# B&R Automation Studio project HISTest (part 4)

```iecst
	SubBMS.Rack4.BSA.Rack_Calc.Field.BRA_Volt_Total 		:=	SHL(DWORD_TO_UINT(SHR(SubBMS.Rack4.BSA.Rack_Calc.Value[0], 8) AND 16#FF), 8) OR	DWORD_TO_UINT(SHR(SubBMS.Rack4.BSA.Rack_Calc.Value[0], 0) AND 16#FF);
	SubBMS.Rack4.BSA.Rack_Calc.Field.BRA_Curr_Total 		:=	SHL(DWORD_TO_UINT(SHR(SubBMS.Rack4.BSA.Rack_Calc.Value[0], 24) AND 16#FF), 8) OR	DWORD_TO_UINT(SHR(SubBMS.Rack4.BSA.Rack_Calc.Value[0], 16) AND 16#FF);
	SubBMS.Rack4.BSA.Rack_Calc.Field.BRA_SOC 				:=	SHL(DWORD_TO_UINT(SHR(SubBMS.Rack4.BSA.Rack_Calc.Value[1], 8) AND 16#FF), 8) OR	DWORD_TO_UINT(SHR(SubBMS.Rack4.BSA.Rack_Calc.Value[1], 0) AND 16#FF);
	SubBMS.Rack4.BSA.Rack_Calc.Field.BRA_SOH 				:=	SHL(DWORD_TO_UINT(SHR(SubBMS.Rack4.BSA.Rack_Calc.Value[1], 24) AND 16#FF), 8) OR	DWORD_TO_UINT(SHR(SubBMS.Rack4.BSA.Rack_Calc.Value[1], 16) AND 16#FF);

	SubBMS.Rack4.BSA.Rack_State.Field.BSA_Divice_Status 	:=	DWORD_TO_USINT(SHR(SubBMS.Rack4.BSA.Rack_State.Value[0], 0) AND 16#0F);
	SubBMS.Rack4.BSA.Rack_State.Field.BSA_Protect_Status 	:=	DWORD_TO_USINT(SHR(SubBMS.Rack4.BSA.Rack_State.Value[0], 8) AND 16#0F);
	SubBMS.Rack4.BSA.Rack_State.Field.BSA_Balance 			:=	SubBMS.Rack4.BSA.Rack_State.Value[0].16;
	SubBMS.Rack4.BSA.Rack_State.Field.BSA_Neg_Rly 			:=	SubBMS.Rack4.BSA.Rack_State.Value[0].17;
	SubBMS.Rack4.BSA.Rack_State.Field.BSA_Pos_Rly 			:=	SubBMS.Rack4.BSA.Rack_State.Value[0].18;
	SubBMS.Rack4.BSA.Rack_State.Field.BSA_PreChar_Rly 		:=	SubBMS.Rack4.BSA.Rack_State.Value[0].19;
	SubBMS.Rack4.BSA.Rack_State.Field.BSA_MSD_AUX 			:=	SubBMS.Rack4.BSA.Rack_State.Value[0].20;
	SubBMS.Rack4.BSA.Rack_State.Field.BSA_EMG_SW 			:=	SubBMS.Rack4.BSA.Rack_State.Value[0].21;
	SubBMS.Rack4.BSA.Rack_State.Field.BSA_Water_leak 		:=	SubBMS.Rack4.BSA.Rack_State.Value[0].22;
	SubBMS.Rack4.BSA.Rack_State.Field.Not_Used1 			:=	SubBMS.Rack4.BSA.Rack_State.Value[0].23;
	SubBMS.Rack4.BSA.Rack_State.Field.Not_Used2 			:=	DWORD_TO_USINT(SHR(SubBMS.Rack4.BSA.Rack_State.Value[0], 24) AND 16#0F);
	SubBMS.Rack4.BSA.Rack_State.Field.BSA_Ah 				:=	SHL(DWORD_TO_UINT(SHR(SubBMS.Rack4.BSA.Rack_State.Value[1], 8) AND 16#FF), 8) OR	DWORD_TO_UINT(SHR(SubBMS.Rack4.BSA.Rack_State.Value[1], 0) AND 16#FF);
	SubBMS.Rack4.BSA.Rack_State.Field.Not_Used3 			:=	SHL(DWORD_TO_UINT(SHR(SubBMS.Rack4.BSA.Rack_State.Value[1], 24) AND 16#FF), 8) OR DWORD_TO_UINT(SHR(SubBMS.Rack4.BSA.Rack_State.Value[1], 16) AND 16#FF);

	SubBMS.Rack4.BSA.Rack_AlarmState.Field.warning.BSA_Wn_Dischager_OC 			:= SubBMS.Rack4.BSA.Rack_AlarmState.Value[0].0;
	SubBMS.Rack4.BSA.Rack_AlarmState.Field.warning.BSA_Wn_Chager_OC				:= SubBMS.Rack4.BSA.Rack_AlarmState.Value[0].1;
	SubBMS.Rack4.BSA.Rack_AlarmState.Field.warning.BSA_Wn_SOC_OV 				:= SubBMS.Rack4.BSA.Rack_AlarmState.Value[0].2;
	SubBMS.Rack4.BSA.Rack_AlarmState.Field.warning.BSA_Wn_SOC_Un  				:= SubBMS.Rack4.BSA.Rack_AlarmState.Value[0].3;
	SubBMS.Rack4.BSA.Rack_AlarmState.Field.warning.BSA_Wn_OV  	 				:= SubBMS.Rack4.BSA.Rack_AlarmState.Value[0].4;
	SubBMS.Rack4.BSA.Rack_AlarmState.Field.warning.BSA_Wn_UV  		 			:= SubBMS.Rack4.BSA.Rack_AlarmState.Value[0].5;
	SubBMS.Rack4.BSA.Rack_AlarmState.Field.warning.BSA_Wn_Cell_OV  				:= SubBMS.Rack4.BSA.Rack_AlarmState.Value[0].6;
	SubBMS.Rack4.BSA.Rack_AlarmState.Field.warning.BSA_Wn_Cell_UV  				:= SubBMS.Rack4.BSA.Rack_AlarmState.Value[0].7;
	SubBMS.Rack4.BSA.Rack_AlarmState.Field.warning.BSA_Wn_Cell_UnbalV  			:= SubBMS.Rack4.BSA.Rack_AlarmState.Value[0].8;
	SubBMS.Rack4.BSA.Rack_AlarmState.Field.warning.BSA_Wn_DisCharger_Cell_OT 	:= SubBMS.Rack4.BSA.Rack_AlarmState.Value[0].9;
	SubBMS.Rack4.BSA.Rack_AlarmState.Field.warning.BSA_Wn_Charger_Cell_OT	 	:= SubBMS.Rack4.BSA.Rack_AlarmState.Value[0].10;
	SubBMS.Rack4.BSA.Rack_AlarmState.Field.warning.BSA_Wn_DisCharger_Cell_UT	:= SubBMS.Rack4.BSA.Rack_AlarmState.Value[0].11;
	SubBMS.Rack4.BSA.Rack_AlarmState.Field.warning.BSA_Wn_Charger_Cell_UT		:= SubBMS.Rack4.BSA.Rack_AlarmState.Value[0].12;
	SubBMS.Rack4.BSA.Rack_AlarmState.Field.warning.BSA_Wn_Cell_UnbalT 			:= SubBMS.Rack4.BSA.Rack_AlarmState.Value[0].13;
	SubBMS.Rack4.BSA.Rack_AlarmState.Field.warning.BSA_Wn_Discharger_UnbaPWR 	:= SubBMS.Rack4.BSA.Rack_AlarmState.Value[0].14;
	SubBMS.Rack4.BSA.Rack_AlarmState.Field.warning.BSA_Wn_Charger_UnbaPWR 		:= SubBMS.Rack4.BSA.Rack_AlarmState.Value[0].15;
	SubBMS.Rack4.BSA.Rack_AlarmState.Field.fault.BSA_FLT_Dischager_OC 			:= SubBMS.Rack4.BSA.Rack_AlarmState.Value[0].16;
	SubBMS.Rack4.BSA.Rack_AlarmState.Field.fault.BSA_FLT_Chager_OC 				:= SubBMS.Rack4.BSA.Rack_AlarmState.Value[0].17;
	SubBMS.Rack4.BSA.Rack_AlarmState.Field.fault.BSA_FLT_SOC_OV  				:= SubBMS.Rack4.BSA.Rack_AlarmState.Value[0].18;
	SubBMS.Rack4.BSA.Rack_AlarmState.Field.fault.BSA_FLT_SOC_Un  				:= SubBMS.Rack4.BSA.Rack_AlarmState.Value[0].19;
	SubBMS.Rack4.BSA.Rack_AlarmState.Field.fault.BSA_FLT_OV  					:= SubBMS.Rack4.BSA.Rack_AlarmState.Value[0].20;
	SubBMS.Rack4.BSA.Rack_AlarmState.Field.fault.BSA_FLT_UV  					:= SubBMS.Rack4.BSA.Rack_AlarmState.Value[0].21;
	SubBMS.Rack4.BSA.Rack_AlarmState.Field.fault.BSA_FLT_Cell_OV  				:= SubBMS.Rack4.BSA.Rack_AlarmState.Value[0].22;
	SubBMS.Rack4.BSA.Rack_AlarmState.Field.fault.BSA_FLT_Cell_UV  				:= SubBMS.Rack4.BSA.Rack_AlarmState.Value[0].23;
	SubBMS.Rack4.BSA.Rack_AlarmState.Field.fault.BSA_FLT_Cell_UnbalV 			:= SubBMS.Rack4.BSA.Rack_AlarmState.Value[0].24;
	SubBMS.Rack4.BSA.Rack_AlarmState.Field.fault.BSA_FLT_DisCharger_Cell_OT  	:= SubBMS.Rack4.BSA.Rack_AlarmState.Value[0].25;
	SubBMS.Rack4.BSA.Rack_AlarmState.Field.fault.BSA_FLT_Charger_Cell_OT  		:= SubBMS.Rack4.BSA.Rack_AlarmState.Value[0].26;
	SubBMS.Rack4.BSA.Rack_AlarmState.Field.fault.BSA_FLT_DisCharger_Cell_UT 	:= SubBMS.Rack4.BSA.Rack_AlarmState.Value[0].27;
	SubBMS.Rack4.BSA.Rack_AlarmState.Field.fault.BSA_FLT_Charger_Cell_UT  		:= SubBMS.Rack4.BSA.Rack_AlarmState.Value[0].28;
	SubBMS.Rack4.BSA.Rack_AlarmState.Field.fault.BSA_FLT_Cell_UnbalT  			:= SubBMS.Rack4.BSA.Rack_AlarmState.Value[0].29;
	SubBMS.Rack4.BSA.Rack_AlarmState.Field.fault.BSA_FLT_Discharger_UnbaPWR  	:= SubBMS.Rack4.BSA.Rack_AlarmState.Value[0].30;
	SubBMS.Rack4.BSA.Rack_AlarmState.Field.fault.BSA_FLT_Charger_UnbaPWR  		:= SubBMS.Rack4.BSA.Rack_AlarmState.Value[0].31;
	SubBMS.Rack4.BSA.Rack_AlarmState.Field.protect.BSA_Prtct_Dischager_OC   	:= SubBMS.Rack4.BSA.Rack_AlarmState.Value[1].0;
	SubBMS.Rack4.BSA.Rack_AlarmState.Field.protect.BSA_Prtct_Chager_OC   		:= SubBMS.Rack4.BSA.Rack_AlarmState.Value[1].1;
	SubBMS.Rack4.BSA.Rack_AlarmState.Field.protect.BSA_Prtct_SOC_OV   		  	:= SubBMS.Rack4.BSA.Rack_AlarmState.Value[1].2;
	SubBMS.Rack4.BSA.Rack_AlarmState.Field.protect.BSA_Prtct_SOC_Un   		  	:= SubBMS.Rack4.BSA.Rack_AlarmState.Value[1].3;
	SubBMS.Rack4.BSA.Rack_AlarmState.Field.protect.BSA_Prtct_OV   		  		:= SubBMS.Rack4.BSA.Rack_AlarmState.Value[1].4;
	SubBMS.Rack4.BSA.Rack_AlarmState.Field.protect.BSA_Prtct_UV   		  		:= SubBMS.Rack4.BSA.Rack_AlarmState.Value[1].5;
	SubBMS.Rack4.BSA.Rack_AlarmState.Field.protect.BSA_Prtct_Cell_OV   		  	:= SubBMS.Rack4.BSA.Rack_AlarmState.Value[1].6;
	SubBMS.Rack4.BSA.Rack_AlarmState.Field.protect.BSA_Prtct_Cell_UV   		  	:= SubBMS.Rack4.BSA.Rack_AlarmState.Value[1].7;
	SubBMS.Rack4.BSA.Rack_AlarmState.Field.protect.BSA_Prtct_Cell_UnbalV   		:= SubBMS.Rack4.BSA.Rack_AlarmState.Value[1].8;
	SubBMS.Rack4.BSA.Rack_AlarmState.Field.protect.BSA_Prtct_DisCharger_Cell_OT := SubBMS.Rack4.BSA.Rack_AlarmState.Value[1].9;
	SubBMS.Rack4.BSA.Rack_AlarmState.Field.protect.BSA_Prtct_Charger_Cell_OT 	:= SubBMS.Rack4.BSA.Rack_AlarmState.Value[1].10;
	SubBMS.Rack4.BSA.Rack_AlarmState.Field.protect.BSA_Prtct_DisCharger_Cell_UT := SubBMS.Rack4.BSA.Rack_AlarmState.Value[1].11;
	SubBMS.Rack4.BSA.Rack_AlarmState.Field.protect.BSA_Prtct_Charger_Cell_UT   	:= SubBMS.Rack4.BSA.Rack_AlarmState.Value[1].12;
	SubBMS.Rack4.BSA.Rack_AlarmState.Field.protect.BSA_Prtct_Cell_UnbalT   		:= SubBMS.Rack4.BSA.Rack_AlarmState.Value[1].13;
	SubBMS.Rack4.BSA.Rack_AlarmState.Field.protect.BSA_Prtct_Discharger_UnbaPWR := SubBMS.Rack4.BSA.Rack_AlarmState.Value[1].14;
	SubBMS.Rack4.BSA.Rack_AlarmState.Field.protect.BSA_Prtct_Charger_UnbaPWR   	:= SubBMS.Rack4.BSA.Rack_AlarmState.Value[1].15;
	SubBMS.Rack4.BSA.Rack_AlarmState.Field.protect.BSA_Prtct_Rly_Err   			:= SubBMS.Rack4.BSA.Rack_AlarmState.Value[1].16;
	SubBMS.Rack4.BSA.Rack_AlarmState.Field.protect.BSA_Prtct_IN_COM_Err   		:= SubBMS.Rack4.BSA.Rack_AlarmState.Value[1].17;
	SubBMS.Rack4.BSA.Rack_AlarmState.Field.protect.BSA_Prtct_EX_COM_Err   		:= SubBMS.Rack4.BSA.Rack_AlarmState.Value[1].18;
	SubBMS.Rack4.BSA.Rack_AlarmState.Field.protect.BSA_Prtct_CT_COM_Err   		:= SubBMS.Rack4.BSA.Rack_AlarmState.Value[1].19;
	SubBMS.Rack4.BSA.Rack_AlarmState.Field.protect.BSA_Prtct_Water_Leak_Err   	:= SubBMS.Rack4.BSA.Rack_AlarmState.Value[1].20;
	SubBMS.Rack4.BSA.Rack_AlarmState.Field.protect.BSA_Prtct_EMS_SW_Err  		:= SubBMS.Rack4.BSA.Rack_AlarmState.Value[1].21;
	SubBMS.Rack4.BSA.Rack_AlarmState.Field.protect.Not_Used1 					:= SubBMS.Rack4.BSA.Rack_AlarmState.Value[1].22;
	SubBMS.Rack4.BSA.Rack_AlarmState.Field.protect.Not_Used2 					:= SubBMS.Rack4.BSA.Rack_AlarmState.Value[1].23;
	SubBMS.Rack4.BSA.Rack_AlarmState.Field.protect.Not_Used3 					:= DWORD_TO_USINT(SHR(SubBMS.Rack4.BSA.Rack_AlarmState.Value[1], 24) AND 16#0F);

	SubBMS.Rack4.BSA.Rack_PWRCalc.Field.BSA_CHAPWCont 							:=	SHL(DWORD_TO_UINT(SHR(SubBMS.Rack4.BSA.Rack_PWRCalc.Value[0], 8) AND 16#FF), 8) OR	DWORD_TO_UINT(SHR(SubBMS.Rack4.BSA.Rack_PWRCalc.Value[0], 0) AND 16#FF);
	SubBMS.Rack4.BSA.Rack_PWRCalc.Field.BSA_DisCHAPWCont 						:=	SHL(DWORD_TO_UINT(SHR(SubBMS.Rack4.BSA.Rack_PWRCalc.Value[0], 24) AND 16#FF), 8) OR	DWORD_TO_UINT(SHR(SubBMS.Rack4.BSA.Rack_PWRCalc.Value[0], 16) AND 16#FF);
	SubBMS.Rack4.BSA.Rack_PWRCalc.Field.BSA_CHAPWPeak 							:=	SHL(DWORD_TO_UINT(SHR(SubBMS.Rack4.BSA.Rack_PWRCalc.Value[1], 8) AND 16#FF), 8) OR	DWORD_TO_UINT(SHR(SubBMS.Rack4.BSA.Rack_PWRCalc.Value[1], 0) AND 16#FF);
	SubBMS.Rack4.BSA.Rack_PWRCalc.Field.BSA_DisCHAPWPeak 						:=	SHL(DWORD_TO_UINT(SHR(SubBMS.Rack4.BSA.Rack_PWRCalc.Value[1], 24) AND 16#FF), 8) OR	DWORD_TO_UINT(SHR(SubBMS.Rack4.BSA.Rack_PWRCalc.Value[1], 16) AND 16#FF);

	SubBMS.Rack4.BSA.Rack_Cell_Vcalc.Field.BSA_Cell_MaxV 						:=	SHL(DWORD_TO_UINT(SHR(SubBMS.Rack4.BSA.Rack_Cell_Vcalc.Value[0], 8) AND 16#FF), 8) OR	DWORD_TO_UINT(SHR(SubBMS.Rack4.BSA.Rack_Cell_Vcalc.Value[0], 0) AND 16#FF);
	SubBMS.Rack4.BSA.Rack_Cell_Vcalc.Field.BSA_Cell_MinV 						:=	SHL(DWORD_TO_UINT(SHR(SubBMS.Rack4.BSA.Rack_Cell_Vcalc.Value[0], 24) AND 16#FF), 8) OR	DWORD_TO_UINT(SHR(SubBMS.Rack4.BSA.Rack_Cell_Vcalc.Value[0], 16) AND 16#FF);
	SubBMS.Rack4.BSA.Rack_Cell_Vcalc.Field.BSA_Cell_AVGV 						:=	SHL(DWORD_TO_UINT(SHR(SubBMS.Rack4.BSA.Rack_Cell_Vcalc.Value[1], 8) AND 16#FF), 8) OR	DWORD_TO_UINT(SHR(SubBMS.Rack4.BSA.Rack_Cell_Vcalc.Value[1], 0) AND 16#FF);
	SubBMS.Rack4.BSA.Rack_Cell_Vcalc.Field.BSA_Cell_DeviV 						:=	SHL(DWORD_TO_UINT(SHR(SubBMS.Rack4.BSA.Rack_Cell_Vcalc.Value[1], 24) AND 16#FF), 8) OR	DWORD_TO_UINT(SHR(SubBMS.Rack4.BSA.Rack_Cell_Vcalc.Value[1], 16) AND 16#FF);

	SubBMS.Rack4.BSA.Rack_Cell_Tcalc.Field.BSA_Cell_MaxT 						:=	SHL(DWORD_TO_UINT(SHR(SubBMS.Rack4.BSA.Rack_Cell_Tcalc.Value[0], 8) AND 16#FF), 8) OR	DWORD_TO_UINT(SHR(SubBMS.Rack4.BSA.Rack_Cell_Tcalc.Value[0], 0) AND 16#FF);
	SubBMS.Rack4.BSA.Rack_Cell_Tcalc.Field.BSA_Cell_MinT 						:=	SHL(DWORD_TO_UINT(SHR(SubBMS.Rack4.BSA.Rack_Cell_Tcalc.Value[0], 24) AND 16#FF), 8) OR	DWORD_TO_UINT(SHR(SubBMS.Rack4.BSA.Rack_Cell_Tcalc.Value[0], 16) AND 16#FF);
	SubBMS.Rack4.BSA.Rack_Cell_Tcalc.Field.BSA_Cell_AVGT 						:=	SHL(DWORD_TO_UINT(SHR(SubBMS.Rack4.BSA.Rack_Cell_Tcalc.Value[1], 8) AND 16#FF), 8) OR	DWORD_TO_UINT(SHR(SubBMS.Rack4.BSA.Rack_Cell_Tcalc.Value[1], 0) AND 16#FF);
	SubBMS.Rack4.BSA.Rack_Cell_Tcalc.Field.BSA_Cell_DeviT 						:=	SHL(DWORD_TO_UINT(SHR(SubBMS.Rack4.BSA.Rack_Cell_Tcalc.Value[1], 24) AND 16#FF), 8) OR	DWORD_TO_UINT(SHR(SubBMS.Rack4.BSA.Rack_Cell_Tcalc.Value[1], 16) AND 16#FF);

	SubBMS.Rack4.BSA.Rack_Cell_Pcalc.Field.BSA_Cell_MaxV_Location 				:=	SHL(DWORD_TO_UINT(SHR(SubBMS.Rack4.BSA.Rack_Cell_Pcalc.Value[0], 8) AND 16#FF), 8) OR	DWORD_TO_UINT(SHR(SubBMS.Rack4.BSA.Rack_Cell_Pcalc.Value[0], 0) AND 16#FF);
	SubBMS.Rack4.BSA.Rack_Cell_Pcalc.Field.BSA_Cell_MinV_Location 				:=	SHL(DWORD_TO_UINT(SHR(SubBMS.Rack4.BSA.Rack_Cell_Pcalc.Value[0], 24) AND 16#FF), 8) OR	DWORD_TO_UINT(SHR(SubBMS.Rack4.BSA.Rack_Cell_Pcalc.Value[0], 16) AND 16#FF);
	SubBMS.Rack4.BSA.Rack_Cell_Pcalc.Field.BSA_Cell_MaxT_Location 				:=	SHL(DWORD_TO_UINT(SHR(SubBMS.Rack4.BSA.Rack_Cell_Pcalc.Value[1], 8) AND 16#FF), 8) OR	DWORD_TO_UINT(SHR(SubBMS.Rack4.BSA.Rack_Cell_Pcalc.Value[1], 0) AND 16#FF);
	SubBMS.Rack4.BSA.Rack_Cell_Pcalc.Field.BSA_Cell_MinT_Location 				:=	SHL(DWORD_TO_UINT(SHR(SubBMS.Rack4.BSA.Rack_Cell_Pcalc.Value[1], 24) AND 16#FF), 8) OR	DWORD_TO_UINT(SHR(SubBMS.Rack4.BSA.Rack_Cell_Pcalc.Value[1], 16) AND 16#FF);

	SubBMS.Rack4.BSA.Modul1_Info.Field.Volt_Total 								:=	SHL(DWORD_TO_UINT(SHR(SubBMS.Rack4.BSA.Modul1_Info.Value[0], 8) AND 16#FF), 8) OR	DWORD_TO_UINT(SHR(SubBMS.Rack4.BSA.Modul1_Info.Value[0], 0) AND 16#FF);
	SubBMS.Rack4.BSA.Modul1_Info.Field.Agv_Volt 								:=	SHL(DWORD_TO_UINT(SHR(SubBMS.Rack4.BSA.Modul1_Info.Value[0], 24) AND 16#FF), 8) OR	DWORD_TO_UINT(SHR(SubBMS.Rack4.BSA.Modul1_Info.Value[0], 16) AND 16#FF);
	SubBMS.Rack4.BSA.Modul1_Info.Field.Agv_Temp 								:=	SHL(DWORD_TO_UINT(SHR(SubBMS.Rack4.BSA.Modul1_Info.Value[1], 8) AND 16#FF), 8) OR	DWORD_TO_UINT(SHR(SubBMS.Rack4.BSA.Modul1_Info.Value[1], 0) AND 16#FF);
	SubBMS.Rack4.BSA.Modul1_Info.Field.OPS_INITOK 								:= SubBMS.Rack4.BSA.Modul1_Info.Value[1].16;
	SubBMS.Rack4.BSA.Modul1_Info.Field.OPS_Fault  								:= SubBMS.Rack4.BSA.Modul1_Info.Value[1].17;
	SubBMS.Rack4.BSA.Modul1_Info.Field.OPS_Balan_On_OFF  						:= SubBMS.Rack4.BSA.Modul1_Info.Value[1].18;
	SubBMS.Rack4.BSA.Modul1_Info.Field.OPS_Waterleak_Err  						:= SubBMS.Rack4.BSA.Modul1_Info.Value[1].19;
	SubBMS.Rack4.BSA.Modul1_Info.Field.OPS_CellVolt_Err  						:= SubBMS.Rack4.BSA.Modul1_Info.Value[1].20;
	SubBMS.Rack4.BSA.Modul1_Info.Field.OPS_CellTemps_Err  						:= SubBMS.Rack4.BSA.Modul1_Info.Value[1].21;
	SubBMS.Rack4.BSA.Modul1_Info.Field.BATIC_Err  								:= SubBMS.Rack4.BSA.Modul1_Info.Value[1].22;
	SubBMS.Rack4.BSA.Modul1_Info.Field.CTCOM_Err  								:= SubBMS.Rack4.BSA.Modul1_Info.Value[1].23;
	SubBMS.Rack4.BSA.Modul1_Info.Field.OPS_MBCOM_Err  							:= SubBMS.Rack4.BSA.Modul1_Info.Value[1].24;
	SubBMS.Rack4.BSA.Modul1_Info.Field.Not_Used1 								:= SubBMS.Rack4.BSA.Modul1_Info.Value[1].25;
	SubBMS.Rack4.BSA.Modul1_Info.Field.Not_Used2  								:= SubBMS.Rack4.BSA.Modul1_Info.Value[1].26;
	SubBMS.Rack4.BSA.Modul1_Info.Field.Not_Used3  								:= SubBMS.Rack4.BSA.Modul1_Info.Value[1].27;
	SubBMS.Rack4.BSA.Modul1_Info.Field.Not_Used4  								:= SubBMS.Rack4.BSA.Modul1_Info.Value[1].28;
	SubBMS.Rack4.BSA.Modul1_Info.Field.Not_Used5  								:= SubBMS.Rack4.BSA.Modul1_Info.Value[1].29;
	SubBMS.Rack4.BSA.Modul1_Info.Field.Not_Used6  								:= SubBMS.Rack4.BSA.Modul1_Info.Value[1].30;
	SubBMS.Rack4.BSA.Modul1_Info.Field.Not_Used7  								:= SubBMS.Rack4.BSA.Modul1_Info.Value[1].31;

	SubBMS.Rack4.BSA.Modul2_Info.Field.Volt_Total 								:=	SHL(DWORD_TO_UINT(SHR(SubBMS.Rack4.BSA.Modul2_Info.Value[0], 8) AND 16#FF), 8) OR	DWORD_TO_UINT(SHR(SubBMS.Rack4.BSA.Modul2_Info.Value[0], 0) AND 16#FF);
	SubBMS.Rack4.BSA.Modul2_Info.Field.Agv_Volt 								:=	SHL(DWORD_TO_UINT(SHR(SubBMS.Rack4.BSA.Modul2_Info.Value[0], 24) AND 16#FF), 8) OR	DWORD_TO_UINT(SHR(SubBMS.Rack4.BSA.Modul2_Info.Value[0], 16) AND 16#FF);
	SubBMS.Rack4.BSA.Modul2_Info.Field.Agv_Temp 								:=	SHL(DWORD_TO_UINT(SHR(SubBMS.Rack4.BSA.Modul2_Info.Value[1], 8) AND 16#FF), 8) OR	DWORD_TO_UINT(SHR(SubBMS.Rack4.BSA.Modul2_Info.Value[1], 0) AND 16#FF);
	SubBMS.Rack4.BSA.Modul2_Info.Field.OPS_INITOK 								:= SubBMS.Rack4.BSA.Modul2_Info.Value[1].16;
	SubBMS.Rack4.BSA.Modul2_Info.Field.OPS_Fault  								:= SubBMS.Rack4.BSA.Modul2_Info.Value[1].17;
	SubBMS.Rack4.BSA.Modul2_Info.Field.OPS_Balan_On_OFF  						:= SubBMS.Rack4.BSA.Modul2_Info.Value[1].18;
	SubBMS.Rack4.BSA.Modul2_Info.Field.OPS_Waterleak_Err  						:= SubBMS.Rack4.BSA.Modul2_Info.Value[1].19;
	SubBMS.Rack4.BSA.Modul2_Info.Field.OPS_CellVolt_Err  						:= SubBMS.Rack4.BSA.Modul2_Info.Value[1].20;
	SubBMS.Rack4.BSA.Modul2_Info.Field.OPS_CellTemps_Err  						:= SubBMS.Rack4.BSA.Modul2_Info.Value[1].21;
	SubBMS.Rack4.BSA.Modul2_Info.Field.BATIC_Err  								:= SubBMS.Rack4.BSA.Modul2_Info.Value[1].22;
	SubBMS.Rack4.BSA.Modul2_Info.Field.CTCOM_Err  								:= SubBMS.Rack4.BSA.Modul2_Info.Value[1].23;
	SubBMS.Rack4.BSA.Modul2_Info.Field.OPS_MBCOM_Err  							:= SubBMS.Rack4.BSA.Modul2_Info.Value[1].24;
	SubBMS.Rack4.BSA.Modul2_Info.Field.Not_Used1 								:= SubBMS.Rack4.BSA.Modul2_Info.Value[1].25;
	SubBMS.Rack4.BSA.Modul2_Info.Field.Not_Used2  								:= SubBMS.Rack4.BSA.Modul2_Info.Value[1].26;
	SubBMS.Rack4.BSA.Modul2_Info.Field.Not_Used3  								:= SubBMS.Rack4.BSA.Modul2_Info.Value[1].27;
	SubBMS.Rack4.BSA.Modul2_Info.Field.Not_Used4  								:= SubBMS.Rack4.BSA.Modul2_Info.Value[1].28;
	SubBMS.Rack4.BSA.Modul2_Info.Field.Not_Used5  								:= SubBMS.Rack4.BSA.Modul2_Info.Value[1].29;
	SubBMS.Rack4.BSA.Modul2_Info.Field.Not_Used6  								:= SubBMS.Rack4.BSA.Modul2_Info.Value[1].30;
	SubBMS.Rack4.BSA.Modul2_Info.Field.Not_Used7  								:= SubBMS.Rack4.BSA.Modul2_Info.Value[1].31;

	SubBMS.Rack4.BSA.Modul3_Info.Field.Volt_Total 								:=	SHL(DWORD_TO_UINT(SHR(SubBMS.Rack4.BSA.Modul3_Info.Value[0], 8) AND 16#FF), 8) OR	DWORD_TO_UINT(SHR(SubBMS.Rack4.BSA.Modul3_Info.Value[0], 0) AND 16#FF);
	SubBMS.Rack4.BSA.Modul3_Info.Field.Agv_Volt 								:=	SHL(DWORD_TO_UINT(SHR(SubBMS.Rack4.BSA.Modul3_Info.Value[0], 24) AND 16#FF), 8) OR	DWORD_TO_UINT(SHR(SubBMS.Rack4.BSA.Modul3_Info.Value[0], 16) AND 16#FF);
	SubBMS.Rack4.BSA.Modul3_Info.Field.Agv_Temp 								:=	SHL(DWORD_TO_UINT(SHR(SubBMS.Rack4.BSA.Modul3_Info.Value[1], 8) AND 16#FF), 8) OR	DWORD_TO_UINT(SHR(SubBMS.Rack4.BSA.Modul3_Info.Value[1], 0) AND 16#FF);
	SubBMS.Rack4.BSA.Modul3_Info.Field.OPS_INITOK 								:= SubBMS.Rack4.BSA.Modul3_Info.Value[1].16;
	SubBMS.Rack4.BSA.Modul3_Info.Field.OPS_Fault  								:= SubBMS.Rack4.BSA.Modul3_Info.Value[1].17;
	SubBMS.Rack4.BSA.Modul3_Info.Field.OPS_Balan_On_OFF  						:= SubBMS.Rack4.BSA.Modul3_Info.Value[1].18;
	SubBMS.Rack4.BSA.Modul3_Info.Field.OPS_Waterleak_Err  						:= SubBMS.Rack4.BSA.Modul3_Info.Value[1].19;
	SubBMS.Rack4.BSA.Modul3_Info.Field.OPS_CellVolt_Err  						:= SubBMS.Rack4.BSA.Modul3_Info.Value[1].20;
	SubBMS.Rack4.BSA.Modul3_Info.Field.OPS_CellTemps_Err  						:= SubBMS.Rack4.BSA.Modul3_Info.Value[1].21;
	SubBMS.Rack4.BSA.Modul3_Info.Field.BATIC_Err  								:= SubBMS.Rack4.BSA.Modul3_Info.Value[1].22;
	SubBMS.Rack4.BSA.Modul3_Info.Field.CTCOM_Err  								:= SubBMS.Rack4.BSA.Modul3_Info.Value[1].23;
	SubBMS.Rack4.BSA.Modul3_Info.Field.OPS_MBCOM_Err  							:= SubBMS.Rack4.BSA.Modul3_Info.Value[1].24;
	SubBMS.Rack4.BSA.Modul3_Info.Field.Not_Used1 								:= SubBMS.Rack4.BSA.Modul3_Info.Value[1].25;
	SubBMS.Rack4.BSA.Modul3_Info.Field.Not_Used2  								:= SubBMS.Rack4.BSA.Modul3_Info.Value[1].26;
	SubBMS.Rack4.BSA.Modul3_Info.Field.Not_Used3  								:= SubBMS.Rack4.BSA.Modul3_Info.Value[1].27;
	SubBMS.Rack4.BSA.Modul3_Info.Field.Not_Used4  								:= SubBMS.Rack4.BSA.Modul3_Info.Value[1].28;
	SubBMS.Rack4.BSA.Modul3_Info.Field.Not_Used5  								:= SubBMS.Rack4.BSA.Modul3_Info.Value[1].29;
	SubBMS.Rack4.BSA.Modul3_Info.Field.Not_Used6  								:= SubBMS.Rack4.BSA.Modul3_Info.Value[1].30;
	SubBMS.Rack4.BSA.Modul3_Info.Field.Not_Used7  								:= SubBMS.Rack4.BSA.Modul3_Info.Value[1].31;

	SubBMS.Rack4.BSA.Modul4_Info.Field.Volt_Total 								:=	SHL(DWORD_TO_UINT(SHR(SubBMS.Rack4.BSA.Modul4_Info.Value[0], 8) AND 16#FF), 8) OR	DWORD_TO_UINT(SHR(SubBMS.Rack4.BSA.Modul4_Info.Value[0], 0) AND 16#FF);
	SubBMS.Rack4.BSA.Modul4_Info.Field.Agv_Volt 								:=	SHL(DWORD_TO_UINT(SHR(SubBMS.Rack4.BSA.Modul4_Info.Value[0], 24) AND 16#FF), 8) OR	DWORD_TO_UINT(SHR(SubBMS.Rack4.BSA.Modul4_Info.Value[0], 16) AND 16#FF);
	SubBMS.Rack4.BSA.Modul4_Info.Field.Agv_Temp 								:=	SHL(DWORD_TO_UINT(SHR(SubBMS.Rack4.BSA.Modul4_Info.Value[1], 8) AND 16#FF), 8) OR	DWORD_TO_UINT(SHR(SubBMS.Rack4.BSA.Modul4_Info.Value[1], 0) AND 16#FF);
	SubBMS.Rack4.BSA.Modul4_Info.Field.OPS_INITOK 								:= SubBMS.Rack4.BSA.Modul4_Info.Value[1].16;
	SubBMS.Rack4.BSA.Modul4_Info.Field.OPS_Fault  								:= SubBMS.Rack4.BSA.Modul4_Info.Value[1].17;
	SubBMS.Rack4.BSA.Modul4_Info.Field.OPS_Balan_On_OFF  						:= SubBMS.Rack4.BSA.Modul4_Info.Value[1].18;
	SubBMS.Rack4.BSA.Modul4_Info.Field.OPS_Waterleak_Err  						:= SubBMS.Rack4.BSA.Modul4_Info.Value[1].19;
	SubBMS.Rack4.BSA.Modul4_Info.Field.OPS_CellVolt_Err  						:= SubBMS.Rack4.BSA.Modul4_Info.Value[1].20;
	SubBMS.Rack4.BSA.Modul4_Info.Field.OPS_CellTemps_Err  						:= SubBMS.Rack4.BSA.Modul4_Info.Value[1].21;
	SubBMS.Rack4.BSA.Modul4_Info.Field.BATIC_Err  								:= SubBMS.Rack4.BSA.Modul4_Info.Value[1].22;
	SubBMS.Rack4.BSA.Modul4_Info.Field.CTCOM_Err  								:= SubBMS.Rack4.BSA.Modul4_Info.Value[1].23;
	SubBMS.Rack4.BSA.Modul4_Info.Field.OPS_MBCOM_Err  							:= SubBMS.Rack4.BSA.Modul4_Info.Value[1].24;
	SubBMS.Rack4.BSA.Modul4_Info.Field.Not_Used1 								:= SubBMS.Rack4.BSA.Modul4_Info.Value[1].25;
	SubBMS.Rack4.BSA.Modul4_Info.Field.Not_Used2  								:= SubBMS.Rack4.BSA.Modul4_Info.Value[1].26;
	SubBMS.Rack4.BSA.Modul4_Info.Field.Not_Used3  								:= SubBMS.Rack4.BSA.Modul4_Info.Value[1].27;
	SubBMS.Rack4.BSA.Modul4_Info.Field.Not_Used4  								:= SubBMS.Rack4.BSA.Modul4_Info.Value[1].28;
	SubBMS.Rack4.BSA.Modul4_Info.Field.Not_Used5  								:= SubBMS.Rack4.BSA.Modul4_Info.Value[1].29;
	SubBMS.Rack4.BSA.Modul4_Info.Field.Not_Used6  								:= SubBMS.Rack4.BSA.Modul4_Info.Value[1].30;
	SubBMS.Rack4.BSA.Modul4_Info.Field.Not_Used7  								:= SubBMS.Rack4.BSA.Modul4_Info.Value[1].31;

	SubBMS.Rack4.BSA.Modul5_Info.Field.Volt_Total 								:=	SHL(DWORD_TO_UINT(SHR(SubBMS.Rack4.BSA.Modul5_Info.Value[0], 8) AND 16#FF), 8) OR	DWORD_TO_UINT(SHR(SubBMS.Rack4.BSA.Modul5_Info.Value[0], 0) AND 16#FF);
	SubBMS.Rack4.BSA.Modul5_Info.Field.Agv_Volt 								:=	SHL(DWORD_TO_UINT(SHR(SubBMS.Rack4.BSA.Modul5_Info.Value[0], 24) AND 16#FF), 8) OR	DWORD_TO_UINT(SHR(SubBMS.Rack4.BSA.Modul5_Info.Value[0], 16) AND 16#FF);
	SubBMS.Rack4.BSA.Modul5_Info.Field.Agv_Temp 								:=	SHL(DWORD_TO_UINT(SHR(SubBMS.Rack4.BSA.Modul5_Info.Value[1], 8) AND 16#FF), 8) OR	DWORD_TO_UINT(SHR(SubBMS.Rack4.BSA.Modul5_Info.Value[1], 0) AND 16#FF);
	SubBMS.Rack4.BSA.Modul5_Info.Field.OPS_INITOK 								:= SubBMS.Rack4.BSA.Modul5_Info.Value[1].16;
	SubBMS.Rack4.BSA.Modul5_Info.Field.OPS_Fault  								:= SubBMS.Rack4.BSA.Modul5_Info.Value[1].17;
	SubBMS.Rack4.BSA.Modul5_Info.Field.OPS_Balan_On_OFF  						:= SubBMS.Rack4.BSA.Modul5_Info.Value[1].18;
	SubBMS.Rack4.BSA.Modul5_Info.Field.OPS_Waterleak_Err  						:= SubBMS.Rack4.BSA.Modul5_Info.Value[1].19;
	SubBMS.Rack4.BSA.Modul5_Info.Field.OPS_CellVolt_Err  						:= SubBMS.Rack4.BSA.Modul5_Info.Value[1].20;
	SubBMS.Rack4.BSA.Modul5_Info.Field.OPS_CellTemps_Err  						:= SubBMS.Rack4.BSA.Modul5_Info.Value[1].21;
	SubBMS.Rack4.BSA.Modul5_Info.Field.BATIC_Err  								:= SubBMS.Rack4.BSA.Modul5_Info.Value[1].22;
	SubBMS.Rack4.BSA.Modul5_Info.Field.CTCOM_Err  								:= SubBMS.Rack4.BSA.Modul5_Info.Value[1].23;
	SubBMS.Rack4.BSA.Modul5_Info.Field.OPS_MBCOM_Err  							:= SubBMS.Rack4.BSA.Modul5_Info.Value[1].24;
	SubBMS.Rack4.BSA.Modul5_Info.Field.Not_Used1 								:= SubBMS.Rack4.BSA.Modul5_Info.Value[1].25;
	SubBMS.Rack4.BSA.Modul5_Info.Field.Not_Used2  								:= SubBMS.Rack4.BSA.Modul5_Info.Value[1].26;
	SubBMS.Rack4.BSA.Modul5_Info.Field.Not_Used3  								:= SubBMS.Rack4.BSA.Modul5_Info.Value[1].27;
	SubBMS.Rack4.BSA.Modul5_Info.Field.Not_Used4  								:= SubBMS.Rack4.BSA.Modul5_Info.Value[1].28;
	SubBMS.Rack4.BSA.Modul5_Info.Field.Not_Used5  								:= SubBMS.Rack4.BSA.Modul5_Info.Value[1].29;
	SubBMS.Rack4.BSA.Modul5_Info.Field.Not_Used6  								:= SubBMS.Rack4.BSA.Modul5_Info.Value[1].30;
	SubBMS.Rack4.BSA.Modul5_Info.Field.Not_Used7  								:= SubBMS.Rack4.BSA.Modul5_Info.Value[1].31;

	SubBMS.Rack4.BSA.Modul6_Info.Field.Volt_Total 								:=	SHL(DWORD_TO_UINT(SHR(SubBMS.Rack4.BSA.Modul6_Info.Value[0], 8) AND 16#FF), 8) OR	DWORD_TO_UINT(SHR(SubBMS.Rack4.BSA.Modul6_Info.Value[0], 0) AND 16#FF);
	SubBMS.Rack4.BSA.Modul6_Info.Field.Agv_Volt 								:=	SHL(DWORD_TO_UINT(SHR(SubBMS.Rack4.BSA.Modul6_Info.Value[0], 24) AND 16#FF), 8) OR	DWORD_TO_UINT(SHR(SubBMS.Rack4.BSA.Modul6_Info.Value[0], 16) AND 16#FF);
	SubBMS.Rack4.BSA.Modul6_Info.Field.Agv_Temp 								:=	SHL(DWORD_TO_UINT(SHR(SubBMS.Rack4.BSA.Modul6_Info.Value[1], 8) AND 16#FF), 8) OR	DWORD_TO_UINT(SHR(SubBMS.Rack4.BSA.Modul6_Info.Value[1], 0) AND 16#FF);
	SubBMS.Rack4.BSA.Modul6_Info.Field.OPS_INITOK 								:= SubBMS.Rack4.BSA.Modul6_Info.Value[1].16;
	SubBMS.Rack4.BSA.Modul6_Info.Field.OPS_Fault  								:= SubBMS.Rack4.BSA.Modul6_Info.Value[1].17;
	SubBMS.Rack4.BSA.Modul6_Info.Field.OPS_Balan_On_OFF  						:= SubBMS.Rack4.BSA.Modul6_Info.Value[1].18;
	SubBMS.Rack4.BSA.Modul6_Info.Field.OPS_Waterleak_Err  						:= SubBMS.Rack4.BSA.Modul6_Info.Value[1].19;
	SubBMS.Rack4.BSA.Modul6_Info.Field.OPS_CellVolt_Err  						:= SubBMS.Rack4.BSA.Modul6_Info.Value[1].20;
	SubBMS.Rack4.BSA.Modul6_Info.Field.OPS_CellTemps_Err  						:= SubBMS.Rack4.BSA.Modul6_Info.Value[1].21;
	SubBMS.Rack4.BSA.Modul6_Info.Field.BATIC_Err  								:= SubBMS.Rack4.BSA.Modul6_Info.Value[1].22;
	SubBMS.Rack4.BSA.Modul6_Info.Field.CTCOM_Err  								:= SubBMS.Rack4.BSA.Modul6_Info.Value[1].23;
	SubBMS.Rack4.BSA.Modul6_Info.Field.OPS_MBCOM_Err  							:= SubBMS.Rack4.BSA.Modul6_Info.Value[1].24;
	SubBMS.Rack4.BSA.Modul6_Info.Field.Not_Used1 								:= SubBMS.Rack4.BSA.Modul6_Info.Value[1].25;
	SubBMS.Rack4.BSA.Modul6_Info.Field.Not_Used2  								:= SubBMS.Rack4.BSA.Modul6_Info.Value[1].26;
	SubBMS.Rack4.BSA.Modul6_Info.Field.Not_Used3  								:= SubBMS.Rack4.BSA.Modul6_Info.Value[1].27;
	SubBMS.Rack4.BSA.Modul6_Info.Field.Not_Used4  								:= SubBMS.Rack4.BSA.Modul6_Info.Value[1].28;
	SubBMS.Rack4.BSA.Modul6_Info.Field.Not_Used5  								:= SubBMS.Rack4.BSA.Modul6_Info.Value[1].29;
	SubBMS.Rack4.BSA.Modul6_Info.Field.Not_Used6  								:= SubBMS.Rack4.BSA.Modul6_Info.Value[1].30;
	SubBMS.Rack4.BSA.Modul6_Info.Field.Not_Used7  								:= SubBMS.Rack4.BSA.Modul6_Info.Value[1].31;

	SubBMS.Rack4.BSA.Modul7_Info.Field.Volt_Total 								:=	SHL(DWORD_TO_UINT(SHR(SubBMS.Rack4.BSA.Modul7_Info.Value[0], 8) AND 16#FF), 8) OR	DWORD_TO_UINT(SHR(SubBMS.Rack4.BSA.Modul7_Info.Value[0], 0) AND 16#FF);
	SubBMS.Rack4.BSA.Modul7_Info.Field.Agv_Volt 								:=	SHL(DWORD_TO_UINT(SHR(SubBMS.Rack4.BSA.Modul7_Info.Value[0], 24) AND 16#FF), 8) OR	DWORD_TO_UINT(SHR(SubBMS.Rack4.BSA.Modul7_Info.Value[0], 16) AND 16#FF);
	SubBMS.Rack4.BSA.Modul7_Info.Field.Agv_Temp 								:=	SHL(DWORD_TO_UINT(SHR(SubBMS.Rack4.BSA.Modul7_Info.Value[1], 8) AND 16#FF), 8) OR	DWORD_TO_UINT(SHR(SubBMS.Rack4.BSA.Modul7_Info.Value[1], 0) AND 16#FF);
	SubBMS.Rack4.BSA.Modul7_Info.Field.OPS_INITOK 								:= SubBMS.Rack4.BSA.Modul7_Info.Value[1].16;
	SubBMS.Rack4.BSA.Modul7_Info.Field.OPS_Fault  								:= SubBMS.Rack4.BSA.Modul7_Info.Value[1].17;
	SubBMS.Rack4.BSA.Modul7_Info.Field.OPS_Balan_On_OFF  						:= SubBMS.Rack4.BSA.Modul7_Info.Value[1].18;
	SubBMS.Rack4.BSA.Modul7_Info.Field.OPS_Waterleak_Err  						:= SubBMS.Rack4.BSA.Modul7_Info.Value[1].19;
	SubBMS.Rack4.BSA.Modul7_Info.Field.OPS_CellVolt_Err  						:= SubBMS.Rack4.BSA.Modul7_Info.Value[1].20;
	SubBMS.Rack4.BSA.Modul7_Info.Field.OPS_CellTemps_Err  						:= SubBMS.Rack4.BSA.Modul7_Info.Value[1].21;
	SubBMS.Rack4.BSA.Modul7_Info.Field.BATIC_Err  								:= SubBMS.Rack4.BSA.Modul7_Info.Value[1].22;
	SubBMS.Rack4.BSA.Modul7_Info.Field.CTCOM_Err  								:= SubBMS.Rack4.BSA.Modul7_Info.Value[1].23;
	SubBMS.Rack4.BSA.Modul7_Info.Field.OPS_MBCOM_Err  							:= SubBMS.Rack4.BSA.Modul7_Info.Value[1].24;
	SubBMS.Rack4.BSA.Modul7_Info.Field.Not_Used1 								:= SubBMS.Rack4.BSA.Modul7_Info.Value[1].25;
	SubBMS.Rack4.BSA.Modul7_Info.Field.Not_Used2  								:= SubBMS.Rack4.BSA.Modul7_Info.Value[1].26;
	SubBMS.Rack4.BSA.Modul7_Info.Field.Not_Used3  								:= SubBMS.Rack4.BSA.Modul7_Info.Value[1].27;
	SubBMS.Rack4.BSA.Modul7_Info.Field.Not_Used4  								:= SubBMS.Rack4.BSA.Modul7_Info.Value[1].28;
	SubBMS.Rack4.BSA.Modul7_Info.Field.Not_Used5  								:= SubBMS.Rack4.BSA.Modul7_Info.Value[1].29;
	SubBMS.Rack4.BSA.Modul7_Info.Field.Not_Used6  								:= SubBMS.Rack4.BSA.Modul7_Info.Value[1].30;
	SubBMS.Rack4.BSA.Modul7_Info.Field.Not_Used7  								:= SubBMS.Rack4.BSA.Modul7_Info.Value[1].31;
END_ACTION
```
